KUKA KRL data list: reinigung.dat

&ACCESS RVO1
&REL 19
&COMMENT Limpeza
&PARAM TEMPLATE = C:\KRC\ROBOTER\TEMPLATE\VG_APPLPROG
&PARAM EDITMASK = *
DEFDAT  REINIGUNG
;FOLD EXTERNAL DECLARATIONS;%{PE}%V3.2.0,%MKUKATPBASIS,%CEXT,%VCOMMON,%P
;FOLD BAS EXT;%{PE}%V3.2.0,%MKUKATPBASIS,%CEXT,%VEXT,%P
EXT  BAS (BAS_COMMAND  :IN,REAL  :IN )
DECL INT SUCCESS
;ENDFOLD
;FOLD A10 EXT;%{E}%V3.2.0,%MKUKATPARC,%CEXT,%VEXT,%P
EXT  A10 (A_CMD_T  :IN,A_STRT_T  :IN,A_WELD_T  :IN,A_END_T  :IN,INT  :IN )
;ENDFOLD
;FOLD A20 EXT;%{E}%V3.2.0,%MKUKATPA20,%CEXT,%VEXT,%P
EXT  A20 (INT  :IN,WELD_ST  :IN,WELD_FI  :IN,INT  :IN )
;ENDFOLD
;FOLD GRIPPER EXT;%{E}%V3.2.0,%MKUKATPGRIPPER,%CEXT,%VEXT,%P
EXT  H50 (INT  :IN,INT  :IN,INT  :IN,GRP_TYP  :IN )
;ENDFOLD
;FOLD SPOT EXT;%{E}%V3.2.0,%MKUKATPSPOT,%CEXT,%VEXT,%P
EXT  USERSPOT (S_COMMAND  :IN,SPOT_TYPE  :IN )
;ENDFOLD
;FOLD TOUCHSENSE EXT;%{E}%V3.2.0,%MKUKATPTS,%CEXT,%VEXT,%P
EXT  H70 (INT  :IN,SRCH_TYP_2  :OUT,E6POS  :IN,SRCH_TYP_3  :IN,SRCH_TYP_2  :IN,SRCH_TYP_2  :IN,SRCH_TYP_2  :IN,SRCH_TYP_2  :IN,SRCH_TYP_2  :IN,INT  :IN )
;ENDFOLD
;FOLD USER EXT;%{E}%V3.2.0,%MKUKATPUSER,%CEXT,%VEXT,%P
;Make here your modifications
;FOLD DC_BOLZEN_V3.01 ;%{}%V3.2.0,%MKUKATPUSER,%CEXT,%VEXT,%P
;EXT  BOLZEN (CALLMODE_T  :IN,INT  :IN,INT  :IN,INT  :IN,INT  :IN )
;ENDFOLD
;FOLD COLLISION_V3.01 ;%{}%V3.2.0,%MKUKATPUSER,%CEXT,%VEXT,%P
EXT  COLLSTOP (INT  :IN,INT  :IN )
;ENDFOLD
;ENDFOLD
;ENDFOLD

DECL BASIS_SUGG_T LAST_BASIS={POINT1[] "P0                      ",POINT2[] "P0                      ",CP_PARAMS[] "CPDAT0                  ",PTP_PARAMS[] "PDAT0                   ",CONT[] "                        ",CP_VEL[] "2                       ",PTP_VEL[] "100                     "}
DECL E6POS XP1={x 2620.46704,y -20.4003601,z 887.235229,a -77.8896179,b 89.3949203,c -77.4276123,s 4,t 24,e1 0.0,e2 0.0,e3 0.0,e4 0.0,e5 0.0,e6 0.0}
DECL E6POS XP2={x 2620.46704,y -20.4003601,z 887.235229,a -77.8896179,b 89.3949203,c -77.4276123,s 4,t 24,e1 0.0,e2 0.0,e3 0.0,e4 0.0,e5 0.0,e6 0.0}
DECL E6POS XWARTUNGSPOS={x 2620.46704,y -20.4003601,z 887.235229,a -77.8896179,b 89.3949203,c -77.4276123,s 4,t 24,e1 0.0,e2 0.0,e3 0.0,e4 0.0,e5 0.0,e6 0.0}
DECL E6POS XP3={x 2620.46704,y -20.4003601,z 887.235229,a -77.8896179,b 89.3949203,c -77.4276123,s 4,t 24,e1 0.0,e2 0.0,e3 0.0,e4 0.0,e5 0.0,e6 0.0}
DECL E6POS XP4={x 2620.46704,y -20.4003601,z 887.235229,a -77.8896179,b 89.3949203,c -77.4276123,s 4,t 24,e1 0.0,e2 0.0,e3 0.0,e4 0.0,e5 0.0,e6 0.0}
DECL E6POS XReinigungsPos={x 802.439819,y 1509.92102,z 316.938812,a -78.5784607,b -42.9682388,c -106.441101,s 2,t 35,e1 0.0,e2 0.0,e3 0.0,e4 0.0,e5 0.0,e6 0.0}
DECL FDAT FP1={TOOL_NO 1,BASE_NO 0,IPO_FRAME #BASE}
DECL PDAT PPDAT={VEL 100.0,ACC 100.0,APO_DIST 100.0}
DECL FDAT FP2={TOOL_NO 1,BASE_NO 0,IPO_FRAME #BASE}
DECL FDAT FWartungsPos={TOOL_NO 1,BASE_NO 0,IPO_FRAME #BASE}
DECL FDAT FP3={TOOL_NO 1,BASE_NO 0,IPO_FRAME #BASE}
DECL FDAT FP4={TOOL_NO 1,BASE_NO 0,IPO_FRAME #BASE}
DECL FDAT FReinigungsPos={TOOL_NO 8,BASE_NO 0,IPO_FRAME #BASE}
ENDDAT
